Yaskawa INFORM job: TESTSFT.JBI

/JOB
//NAME TESTSFT
//POS
///NPOS 3,3,0,2,0,0
///TOOL 0
///POSTYPE ROBOT
///RECTAN
///RCONF 0,0,0,0,0,0,0,0,0,0,0,0,0,0,0,0,0,0,0,0,0,0,0,0
C00000=1313.963,-672.963,-1888.710,-38.6808,29.6683,56.1213
C00001=1313.963,-672.963,-1888.710,-38.6808,29.6683,56.1213
C00002=1313.963,-672.963,-1888.710,-38.6808,29.6683,56.1213
BC00000=385.112,2573.309,1636.940
BC00001=385.112,2573.309,1636.940
BC00002=385.112,2573.309,1636.940
///POSTYPE BASE
P00300=10.000,0.000,15.000,0.0000,0.0000,0.0000
P00301=-10.000,0.000,20.000,0.0000,0.0000,0.0000
//INST
///DATE 2024/02/07 19:56
///ATTR SC,RW,RJ
////FRAME ROBOT
///GROUP1 RB1,BS1
NOP
SFTOF
MOVL C00000 BC00000 V=20.0
SFTON P300
MOVL C00001 BC00001 V=20.0
PAUSE
SFTON P301
MOVL C00002 BC00002 V=20.0
PAUSE
SFTOF
END
